FUNCTION_BLOCK FB_WriteChange_STR
VAR_INPUT
	i_bScan			:BOOL;
	i_bWrite		:BOOL;
	i_sVar			:STRING;
	i_enEvent		:EN_BatchEvents;
	i_sDescription	:STRING;
END_VAR
VAR
	sVarOld			:STRING;
	bVarOld			:BOOL;
	Trig			:R_TRIG;
	bScan			:BOOL;
	Scan_TON		:TON;
END_VAR
VAR_IN_OUT
	iq_stParams		:ST_AuditTrail;
	iq_bWrite		:BOOL;
END_VAR

IF i_bScan THEN
	bScan:=TRUE;
END_IF
Scan_TON(IN:=bScan,PT:=T#1S);
IF Scan_TON.Q THEN
	sVarOld:=i_sVar;
	bScan:=FALSE;
END_IF
Trig(CLK:=i_bWrite);
IF Trig.Q AND NOT bScan THEN
	iq_stParams.Event:=TO_STRING(i_enEvent);
	iq_stParams.Description := i_sDescription;
	iq_stParams.Oldvalue:=sVarOld;
	iq_stParams.Newvalue:=i_sVar;
	sVarOld:=i_sVar;
	iq_bWrite:=TRUE;
END_IF

END_FUNCTION_BLOCK

(* stored: Version 1.1.0.1, ProductVersion 3.1.4024.12
   POU FB_WriteChange_STR: Id {951b0762-feda-44e5-b3b7-f7874ce926b3}, SpecialFunc None *)
